PROGRAM MAIN
VAR

END_VAR

PRG_Schrauber();

END_PROGRAM

(* stored: Version 1.1.0.1, ProductVersion 3.1.4024.15
   POU MAIN: Id {2cd6c072-ca5e-4bc3-9fe1-6217351787c7}, SpecialFunc None *)
